VAR_GLOBAL CONSTANT
	/// max size of lookup table
	MaxLookupSize: INT := 30;
END_VAR

(* stored: Version 1.1.0.1, ProductVersion 3.1.0.36
   GVL LUT_Constants: Id {af67a2b8-ca5f-44b6-8761-347846921ecc} *)
